// TIA Portal project "2020-11-20_LampeggioPlus" (V16)
// Programma che gestisce la ventilazione di un motore

(* hardware
DEVICE "Stazione SIMATIC 1200_1"  S71200.Device
   slot 0: "Telaio di montaggio S7-1200"  Rack  V1.0
   slot 1: "PLC_1"  CPU 1215C DC/DC/DC  6ES7 215-1AG40-0XB0  V4.2
*)

// ===== PLC "PLC_1"  CPU 1215C DC/DC/DC =====

VAR_GLOBAL   // PLC tag table "Tabella delle variabili standard"
   "in0_f" AT %I0.0 : Bool;
   "in1_f" AT %I0.1 : Bool;
   "in2_f" AT %I0.2 : Bool;
   "in3_f" AT %I0.3 : Bool;
   "in4_f" AT %I0.4 : Bool;
   "in5_f" AT %I0.5 : Bool;
   "in6_f" AT %I0.6 : Bool;
   "led" AT %Q0.7 : Bool;
   "errore switch" AT %Q0.1 : Bool;
   "in7_f" AT %I0.7 : Bool;
   "out2" AT %Q0.2 : Bool;
   "out3" AT %Q0.3 : Bool;
   "out4" AT %Q0.4 : Bool;
   "sempre vero" AT %M6.0 : Bool;   // bit sempre vero
   "uscite byte" AT %QB0 : Byte;   // Uscite fisiche
   "uscite memorie" AT %MB1 : Byte;   // uscite memorie da usare come ingressi
   "out4_M" AT %M1.4 : Bool;
   "out3_M" AT %M1.3 : Bool;
   "out2_M" AT %M1.2 : Bool;
   "errore switch_M" AT %M1.1 : Bool;
   "led_M" AT %M1.7 : Bool;
   "ingressi byte" AT %IB0 : Byte;   // Ingressi fisici
   "ingressi memorie" AT %MB0 : Byte;   // Ingressi Na non filtrati
   "in0_na" AT %M0.0 : Bool;
   "in1_na" AT %M0.1 : Bool;
   "in2_na" AT %M0.2 : Bool;
   "in3_na" AT %M0.3 : Bool;
   "in4_na" AT %M0.4 : Bool;
   "in5_na" AT %M0.5 : Bool;
   "in6_na" AT %M0.6 : Bool;
   "in7_na" AT %M0.7 : Bool;
   "out5" AT %Q0.5 : Bool;
   "out6" AT %Q0.6 : Bool;
   "out0" AT %Q0.0 : Bool;
   "out5_M" AT %M1.5 : Bool;
   "out6_M" AT %M1.6 : Bool;
   "out7_M" AT %M1.0 : Bool;
   "ingressi memorie filtrato" AT %MB2 : Byte;
   "Abil_S" AT %M2.1 : Bool;
   "Abil_A" AT %M2.0 : Bool;
   "Abil_Val" AT %M2.2 : Bool;
   "in3" AT %M2.3 : Bool;
   "Val_lsb" AT %M2.4 : Bool;
   "Val_2" AT %M2.5 : Bool;
   "Val_3" AT %M2.6 : Bool;
   "Val_4" AT %M2.7 : Bool;
   "ingressi memorie_p" AT %MB3 : Byte;
   "Abil_S_p" AT %M3.1 : Bool;   // finecorsa di sicurezza
   "Abil_A_p" AT %M3.0 : Bool;   // presenza tensione al motore
   "Abil_Val_p" AT %M3.2 : Bool;   // presenza Allarme
   "in3_p" AT %M3.3 : Bool;   // ventilazione motore ON
   "in4_p" AT %M3.4 : Bool;   // motore troppo caldo
   "in5_p" AT %M3.5 : Bool;   // comando avviamento motore
   "in6_p" AT %M3.6 : Bool;   // comando arresto motore
   "in7_p" AT %M3.7 : Bool;   // Reset memorizzazione Allarme
   "ingressi_memorie_var_p" AT %MB4 : Byte;
   "in0_var_p" AT %M4.0 : Bool;   // finecorsa di sicurezza
   "in1_var_p" AT %M4.1 : Bool;   // presenza tensione al motore
   "in2_var_p" AT %M4.2 : Bool;   // presenza Allarme
   "in3_var_p" AT %M4.3 : Bool;   // ventilazione motore ON
   "in4_var_p" AT %M4.4 : Bool;   // motore troppo caldo
   "in5_var_p" AT %M4.5 : Bool;   // comando avviamento motore
   "in6_var_p" AT %M4.6 : Bool;   // comando arresto motore
   "in7_var_p" AT %M4.7 : Bool;   // Reset memorizzazione Allarme
   "Semiperiodo" AT %MD20 : Time;
   "Var_Byte" AT %MB24 : Byte;
END_VAR

VAR_GLOBAL CONSTANT   // PLC tag table "Tabella delle variabili standard"
   "maschera NCNA" : Byte := B#2#00000000;   // mettere a 1 i bit NC
   "filtro in0" : Time := T#200ms;
   "filtro in1" : Time := T#200ms;
   "filtro in2" : Time := T#1s;
   "filtro in3" : Time := T#200ms;
   "filtro in4" : Time := T#1s;
   "filtro in5" : Time := T#1s;
   "filtro in6" : Time := T#1s;
   "filtro in7" : Time := T#1s;
   "Maschera Out Reset" : Byte := B#2#00000000;
   "Maschera Val" : Byte := B#2#11110000;
   "Numero_Shift" : Byte := 4;
   "Tempo_fisso_lampeggio" : Time := T#1s;
   "Tempo_quanto_x_mul" : Time := T#100ms;
END_VAR

// folder: System blocks/Program resources

DATA_BLOCK "filtro_in0"   // DB1
{ S7_Optimized_Access := 'TRUE' }
AUTHOR : Simatic
FAMILY : IEC
NAME : IEC_TMR
VERSION : 1.0
// stored: InstanceOfName IEC_TIMER
"IEC_TIMER"
BEGIN
END_DATA_BLOCK

DATA_BLOCK "filtro_in1"   // DB2
{ S7_Optimized_Access := 'TRUE' }
AUTHOR : Simatic
FAMILY : IEC
NAME : IEC_TMR
VERSION : 1.0
// stored: InstanceOfName IEC_TIMER
"IEC_TIMER"
BEGIN
END_DATA_BLOCK

DATA_BLOCK "filtro_in2"   // DB3
{ S7_Optimized_Access := 'TRUE' }
AUTHOR : Simatic
FAMILY : IEC
NAME : IEC_TMR
VERSION : 1.0
// stored: InstanceOfName IEC_TIMER
"IEC_TIMER"
BEGIN
END_DATA_BLOCK

DATA_BLOCK "filtro_in3"   // DB4
{ S7_Optimized_Access := 'TRUE' }
AUTHOR : Simatic
FAMILY : IEC
NAME : IEC_TMR
VERSION : 1.0
// stored: InstanceOfName IEC_TIMER
"IEC_TIMER"
BEGIN
END_DATA_BLOCK

DATA_BLOCK "filtro_in4"   // DB5
{ S7_Optimized_Access := 'TRUE' }
AUTHOR : Simatic
FAMILY : IEC
NAME : IEC_TMR
VERSION : 1.0
// stored: InstanceOfName IEC_TIMER
"IEC_TIMER"
BEGIN
END_DATA_BLOCK

DATA_BLOCK "filtro_in5"   // DB6
{ S7_Optimized_Access := 'TRUE' }
AUTHOR : Simatic
FAMILY : IEC
NAME : IEC_TMR
VERSION : 1.0
// stored: InstanceOfName IEC_TIMER
"IEC_TIMER"
BEGIN
END_DATA_BLOCK

DATA_BLOCK "filtro_in6"   // DB7
{ S7_Optimized_Access := 'TRUE' }
AUTHOR : Simatic
FAMILY : IEC
NAME : IEC_TMR
VERSION : 1.0
// stored: InstanceOfName IEC_TIMER
"IEC_TIMER"
BEGIN
END_DATA_BLOCK

DATA_BLOCK "filtro_in7"   // DB8
{ S7_Optimized_Access := 'TRUE' }
AUTHOR : Simatic
FAMILY : IEC
NAME : IEC_TMR
VERSION : 1.0
// stored: InstanceOfName IEC_TIMER
"IEC_TIMER"
BEGIN
END_DATA_BLOCK

DATA_BLOCK "timer_toff"   // DB9
{ S7_Optimized_Access := 'TRUE' }
AUTHOR : Simatic
FAMILY : IEC
NAME : IEC_TMR
VERSION : 1.0
// stored: InstanceOfName IEC_TIMER
"IEC_TIMER"
BEGIN
END_DATA_BLOCK

DATA_BLOCK "timer_ton"   // DB10
{ S7_Optimized_Access := 'TRUE' }
AUTHOR : Simatic
FAMILY : IEC
NAME : IEC_TMR
VERSION : 1.0
// stored: InstanceOfName IEC_TIMER
"IEC_TIMER"
BEGIN
END_DATA_BLOCK

// folder: (top level)

FUNCTION "Ingressi e uscite" : Void   // FC1, LAD
{ S7_Optimized_Access := 'TRUE' }
VERSION : 0.1
   VAR_TEMP   // added for the SCL form of the ladder/FBD networks
      _w1 : Bool;
   END_VAR
BEGIN

REGION Network 1: creazione immagine uscite (MB1) da usare come ingressi
   // creazione immagine uscite (MB1) da usare come ingressi
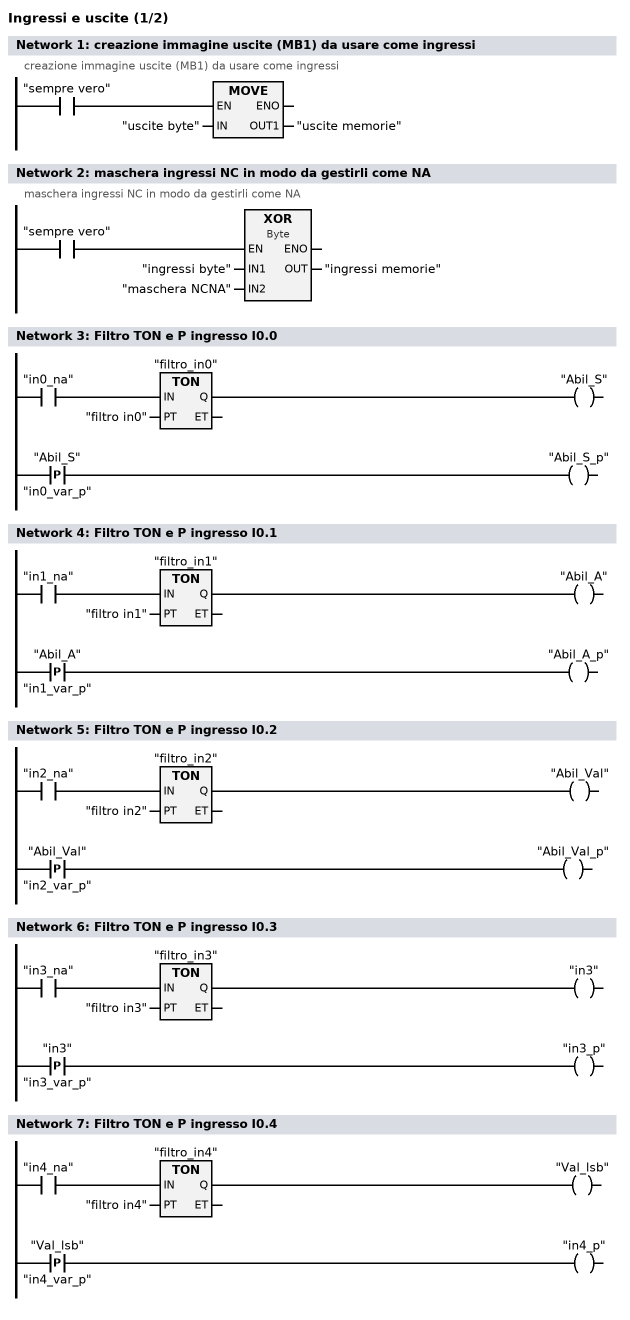
   RUNG wire#powerrail
      Contact( "sempre vero" )
      { S7_GenerateENO := "TRUE" } Move(in := "uscite byte", out1 => "uscite memorie")
   END_RUNG
   // the same network as SCL:
   IF "sempre vero" THEN "uscite memorie" := "uscite byte"; END_IF;
END_REGION

REGION Network 2: maschera ingressi NC in modo da gestirli come NA
   // maschera ingressi NC in modo da gestirli come NA
   IF "sempre vero" THEN "ingressi memorie" := "ingressi byte" XOR "maschera NCNA"; END_IF;
END_REGION

REGION Network 3: Filtro TON e P ingresso I0.0
   "filtro_in0".TON(IN := "in0_na", PT := "filtro in0");
   "Abil_S" := "filtro_in0".Q;
   #_w1 := "Abil_S" AND NOT "in0_var_p";   // rising edge of "Abil_S"
   "in0_var_p" := "Abil_S";
   "Abil_S_p" := #_w1;
END_REGION

REGION Network 4: Filtro TON e P ingresso I0.1
   "filtro_in1".TON(IN := "in1_na", PT := "filtro in1");
   "Abil_A" := "filtro_in1".Q;
   #_w1 := "Abil_A" AND NOT "in1_var_p";   // rising edge of "Abil_A"
   "in1_var_p" := "Abil_A";
   "Abil_A_p" := #_w1;
END_REGION

REGION Network 5: Filtro TON e P ingresso I0.2
   "filtro_in2".TON(IN := "in2_na", PT := "filtro in2");
   "Abil_Val" := "filtro_in2".Q;
   #_w1 := "Abil_Val" AND NOT "in2_var_p";   // rising edge of "Abil_Val"
   "in2_var_p" := "Abil_Val";
   "Abil_Val_p" := #_w1;
END_REGION

REGION Network 6: Filtro TON e P ingresso I0.3
   "filtro_in3".TON(IN := "in3_na", PT := "filtro in3");
   "in3" := "filtro_in3".Q;
   #_w1 := "in3" AND NOT "in3_var_p";   // rising edge of "in3"
   "in3_var_p" := "in3";
   "in3_p" := #_w1;
END_REGION

REGION Network 7: Filtro TON e P ingresso I0.4
   "filtro_in4".TON(IN := "in4_na", PT := "filtro in4");
   "Val_lsb" := "filtro_in4".Q;
   #_w1 := "Val_lsb" AND NOT "in4_var_p";   // rising edge of "Val_lsb"
   "in4_var_p" := "Val_lsb";
   "in4_p" := #_w1;
END_REGION

REGION Network 8: Filtro TON e P ingresso I0.5
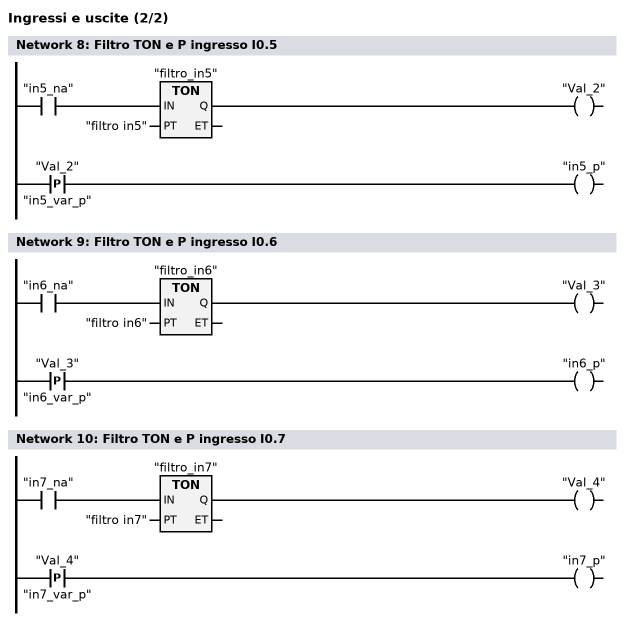
   "filtro_in5".TON(IN := "in5_na", PT := "filtro in5");
   "Val_2" := "filtro_in5".Q;
   #_w1 := "Val_2" AND NOT "in5_var_p";   // rising edge of "Val_2"
   "in5_var_p" := "Val_2";
   "in5_p" := #_w1;
END_REGION

REGION Network 9: Filtro TON e P ingresso I0.6
   "filtro_in6".TON(IN := "in6_na", PT := "filtro in6");
   "Val_3" := "filtro_in6".Q;
   #_w1 := "Val_3" AND NOT "in6_var_p";   // rising edge of "Val_3"
   "in6_var_p" := "Val_3";
   "in6_p" := #_w1;
END_REGION

REGION Network 10: Filtro TON e P ingresso I0.7
   "filtro_in7".TON(IN := "in7_na", PT := "filtro in7");
   "Val_4" := "filtro_in7".Q;
   #_w1 := "Val_4" AND NOT "in7_var_p";   // rising edge of "Val_4"
   "in7_var_p" := "Val_4";
   "in7_p" := #_w1;
END_REGION
END_FUNCTION

FUNCTION "Calcolo_Tempo" : Void   // FC2, LAD
{ S7_Optimized_Access := 'TRUE' }
VERSION : 0.1
// Utilizza:
// MB2  Ingressi memorie filtrato
// M2.2 Abil_lampeggio a tempo variabile
// MD20  semiperiodo
// MB24 Variabile Byte temporanea
// Valori costanti
BEGIN

REGION Network 1
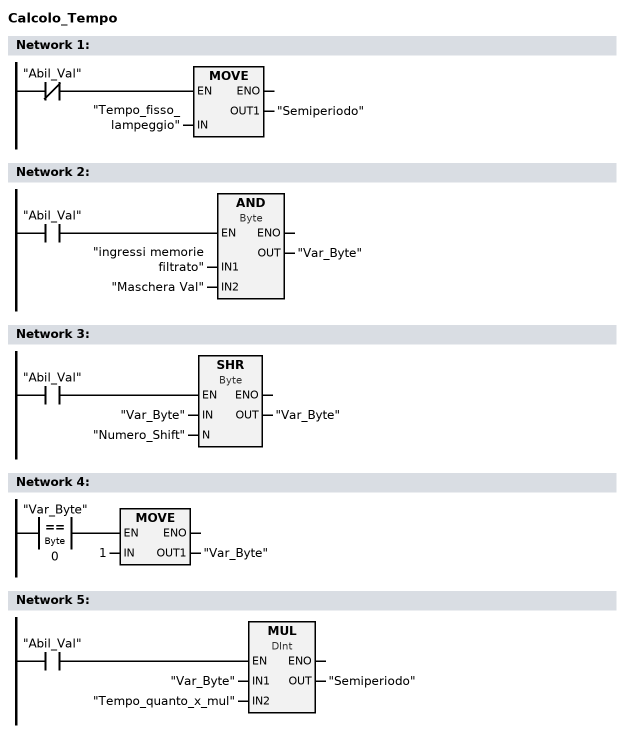
   RUNG wire#powerrail
      I_Contact( "Abil_Val" )
      { S7_GenerateENO := "TRUE" } Move(in := "Tempo_fisso_lampeggio", out1 => "Semiperiodo")
   END_RUNG
   // the same network as SCL:
   IF NOT "Abil_Val" THEN "Semiperiodo" := "Tempo_fisso_lampeggio"; END_IF;
END_REGION

REGION Network 2
   RUNG wire#powerrail
      Contact( "Abil_Val" )
      { S7_Templates := "SrcType := Byte"; S7_GenerateENO := "TRUE" } And(in1 := "ingressi memorie filtrato", in2 := "Maschera Val", out => "Var_Byte")
   END_RUNG
   // the same network as SCL:
   IF "Abil_Val" THEN "Var_Byte" := "ingressi memorie filtrato" AND "Maschera Val"; END_IF;
END_REGION

REGION Network 3
   RUNG wire#powerrail
      Contact( "Abil_Val" )
      { S7_Templates := "SrcType := Byte"; S7_GenerateENO := "TRUE" } Shr(in := "Var_Byte", n := "Numero_Shift", out => "Var_Byte")
   END_RUNG
   // the same network as SCL:
   IF "Abil_Val" THEN "Var_Byte" := SHR(IN := "Var_Byte", N := "Numero_Shift"); END_IF;
END_REGION

REGION Network 4
   RUNG wire#powerrail
      { S7_Templates := "SrcType := Byte" } EQ_Contact(in1 := "Var_Byte", in2 := 0)
      { S7_GenerateENO := "TRUE" } Move(in := 1, out1 => "Var_Byte")
   END_RUNG
   // the same network as SCL:
   IF "Var_Byte" = 0 THEN "Var_Byte" := 1; END_IF;
END_REGION

REGION Network 5
   RUNG wire#powerrail
      Contact( "Abil_Val" )
      { S7_Templates := "SrcType := DInt"; S7_GenerateENO := "TRUE" } Mul(in1 := "Var_Byte", in2 := "Tempo_quanto_x_mul", out => "Semiperiodo")
   END_RUNG
   // the same network as SCL:
   IF "Abil_Val" THEN "Semiperiodo" := "Var_Byte" * "Tempo_quanto_x_mul"; END_IF;
END_REGION
END_FUNCTION

ORGANIZATION_BLOCK "Main"   // OB1, LAD, ProgramCycle
TITLE = "Main Program Sweep (Cycle)"
{ S7_Optimized_Access := 'TRUE' }
VERSION : 0.1
// Programma che fa Lampeggiare Q0.7 a frequenza di 0,5Hz se Abil_Val (I0.2, NA, 200ms ) è off, mentre il semiperiodo di lampeggio è pari a 100ms*NUM dove NUM è il numero binario da 1 a 15 formato dai bit I0.4-I0.7 (tutti NA, 1s).
// Il lampeggio parte da acceso se va a 1 Abil_A (I0.0, NA, 200ms) e parte da spento se va a 1 Abil_S (I0.1, NA, 200ms).
// Segnalazione di errore su Q0.1 se I0.4-I0.7=0000 e limite a 1 per NUM
// 
// 
// Programma 8_programma base
// predisposizione ingressi con compensazione NC e filtro di ritardo all'inserzione. Generazione OB100 (Startup) per reset uscite e variabili)
BEGIN

REGION Network 1: richiamo FC Ingressi Uscite
   // creazione immagine uscite (MB1) da usare come ingressi
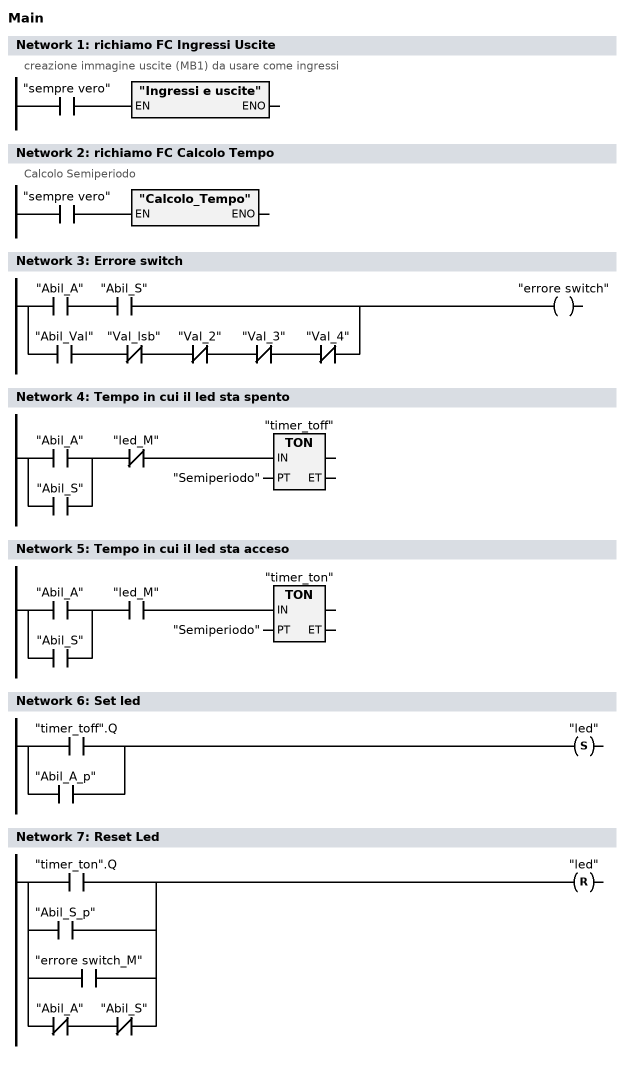
   RUNG wire#powerrail
      Contact( "sempre vero" )
      "Ingressi e uscite"()
   END_RUNG
   // the same network as SCL:
   IF "sempre vero" THEN "Ingressi e uscite"(); END_IF;
END_REGION

REGION Network 2: richiamo FC Calcolo Tempo
   // Calcolo Semiperiodo
   RUNG wire#powerrail
      Contact( "sempre vero" )
      "Calcolo_Tempo"()
   END_RUNG
   // the same network as SCL:
   IF "sempre vero" THEN "Calcolo_Tempo"(); END_IF;
END_REGION

REGION Network 3: Errore switch
   RUNG wire#powerrail
      Contact( "Abil_A" )
      Contact( "Abil_S" )
      wire#w1
      Coil( "errore switch" )
   END_RUNG
   RUNG wire#powerrail
      Contact( "Abil_Val" )
      I_Contact( "Val_lsb" )
      I_Contact( "Val_2" )
      I_Contact( "Val_3" )
      I_Contact( "Val_4" )
   END_RUNG wire#w1
   // the same network as SCL:
   "errore switch" := ("Abil_A" AND "Abil_S") OR ("Abil_Val" AND NOT "Val_lsb" AND NOT "Val_2" AND NOT "Val_3" AND NOT "Val_4");
END_REGION

REGION Network 4: Tempo in cui il led sta spento
   "timer_toff".TON(IN := ("Abil_A" OR "Abil_S") AND NOT "led_M", PT := "Semiperiodo");
END_REGION

REGION Network 5: Tempo in cui il led sta acceso
   "timer_ton".TON(IN := ("Abil_A" OR "Abil_S") AND "led_M", PT := "Semiperiodo");
END_REGION

REGION Network 6: Set led
   RUNG wire#powerrail
      Contact( "timer_toff".Q )
      wire#w1
      S_Coil( "led" )
   END_RUNG
   RUNG wire#powerrail
      Contact( "Abil_A_p" )
   END_RUNG wire#w1
   // the same network as SCL:
   IF "timer_toff".Q OR "Abil_A_p" THEN "led" := TRUE; END_IF;
END_REGION

REGION Network 7: Reset Led
   RUNG wire#powerrail
      Contact( "timer_ton".Q )
      wire#w1
      R_Coil( "led" )
   END_RUNG
   RUNG wire#powerrail
      Contact( "Abil_S_p" )
   END_RUNG wire#w1
   RUNG wire#powerrail
      Contact( "errore switch_M" )
   END_RUNG wire#w1
   RUNG wire#powerrail
      I_Contact( "Abil_A" )
      I_Contact( "Abil_S" )
   END_RUNG wire#w1
   // the same network as SCL:
   IF "timer_ton".Q OR "Abil_S_p" OR "errore switch_M" OR (NOT "Abil_A" AND NOT "Abil_S") THEN
       "led" := FALSE;
   END_IF;
END_REGION
END_ORGANIZATION_BLOCK

ORGANIZATION_BLOCK "Startup"   // OB100, LAD, Startup
TITLE = "Complete Restart"
{ S7_Optimized_Access := 'TRUE' }
VERSION : 0.1
   VAR_INPUT
      LostRetentive : Bool;   // True if retentive data are lost
      LostRTC : Bool;   // True if real time clock is lost
   END_VAR
BEGIN

REGION Network 1: bit sempre vero
   // creazione bit sempre vero
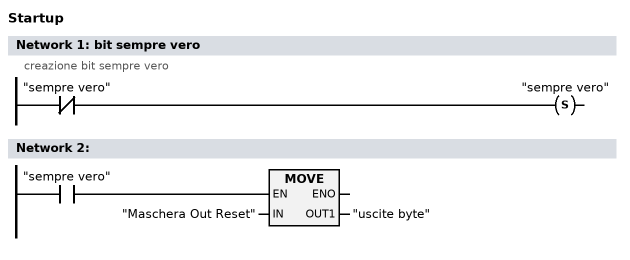
   RUNG wire#powerrail
      I_Contact( "sempre vero" )
      S_Coil( "sempre vero" )
   END_RUNG
   // the same network as SCL:
   IF NOT "sempre vero" THEN "sempre vero" := TRUE; END_IF;
END_REGION

REGION Network 2
   RUNG wire#powerrail
      Contact( "sempre vero" )
      { S7_GenerateENO := "TRUE" } Move(in := "Maschera Out Reset", out1 => "uscite byte")
   END_RUNG
   // the same network as SCL:
   IF "sempre vero" THEN "uscite byte" := "Maschera Out Reset"; END_IF;
END_REGION
END_ORGANIZATION_BLOCK